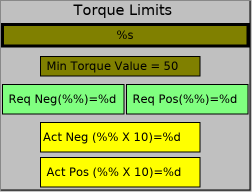
VISUALIZATION TORQUE  // 252x192
VAR_INPUT
	{attribute 'parameterstringof' := 'm_Input_Instance'}
	m_Input_Instance_Str : STRING;
END_VAR
VAR_IN_OUT
	m_Input_Instance : None;
END_VAR
    Rectangle (0,0 250x190), "Torque Limits"
    RoundedRectangle (2,84 122x30), "Req Neg(%%)=%d", text variable: Global_Var_AxisInterface.stAxesGlobalVars[m_Input_Instance].stTorque.NegReq, input disabled if: Global_Var_AxisInterface.AxesfunctionsVisDisable
        OnMouseDown: write the text variable via Edit, min 1, max 100
    RoundedRectangle (126,84 122x30), "Req Pos(%%)=%d", text variable: Global_Var_AxisInterface.stAxesGlobalVars[m_Input_Instance].stTorque.PosReq, input disabled if: Global_Var_AxisInterface.AxesfunctionsVisDisable
        OnMouseDown: write the text variable via Edit, min 1, max 100
    RoundedRectangle (40,122 160x30), "Act Neg (%% X 10)=%d", text variable: Global_Var_AxisInterface.stDriveOut[m_Input_Instance].TorqueNeg
    RoundedRectangle (40,157 160x30), "Act Pos (%% X 10)=%d", text variable: Global_Var_AxisInterface.stDriveOut[m_Input_Instance].TorquePos
    RoundedRectangle (40,56 160x20), "Min Torque Value = 50"
    Rectangle (1,23 248x24), "%s", text variable: m_Input_Instance_Str
END_VISUALIZATION

(* stored: Version 1.1.0.1, ProductVersion 3.1.4024.11
   Visu TORQUE: Id {4e8c74af-b480-43bd-8ff4-51b7aebb12b8} *)
